TYPE EStatus :
(
	NotReady,
	Ready,
	Prefilling,
	DeliverLiquid,
	Error,
	PreparingForNextDrink,
	MeasuringContent,
	RunningManualDeliver
);
END_TYPE

(* stored: Version 1.1.0.1, ProductVersion 3.1.0.19
   DUT EStatus: Id {4a12072d-8be6-4bb2-9c5a-12e69b424b19} *)
